// TIA Portal project "Fase_4" (V17)

(* hardware
DEVICE "S7-1200 station_1"  S7-1200 Station
   slot 0: "Rack_0"  S7-1200 Rack  Rack  V1.0
   slot 1: "PLC_1"  CPU 1214C AC/DC/Rly  6ES7 214-1BE30-0XB0  V2.2
*)

// ===== PLC "PLC_1"  CPU 1214C AC/DC/Rly =====

VAR_GLOBAL   // PLC tag table "Default tag table"
   "aumentarcoches" AT %M100.0 : Bool;
   "quitarcoches" AT %M100.1 : Bool;
   "Tag_1" AT %M202.2 : Bool;
   "Tag_2" AT %MW320 : Int;
   "Tag_3" AT %MW420 : Int;
   "verde" AT %M1.0 : Bool;
   "naranja" AT %M1.1 : Bool;
   "rojo" AT %M1.2 : Bool;
END_VAR

// folder: System blocks/Program resources

DATA_BLOCK "numerocoches"   // DB1
{ S7_Optimized_Access := 'TRUE' }
AUTHOR : Simatic
FAMILY : IEC
NAME : CNTR
VERSION : 1.0
// stored: InstanceOfName IEC_COUNTER
"IEC_COUNTER"
BEGIN
END_DATA_BLOCK

// folder: (top level)

ORGANIZATION_BLOCK "Main"   // OB1, LAD, ProgramCycle
TITLE = "Main Program Sweep (Cycle)"
{ S7_Optimized_Access := 'TRUE' }
VERSION : 0.1
// Es un garaje monitorizado.
BEGIN

REGION Network 1
   // Esto es un contador de coches, M100 aumenta en uno el numero de coches, M100.1 quita un coche y MW320  recoge el numero de coches
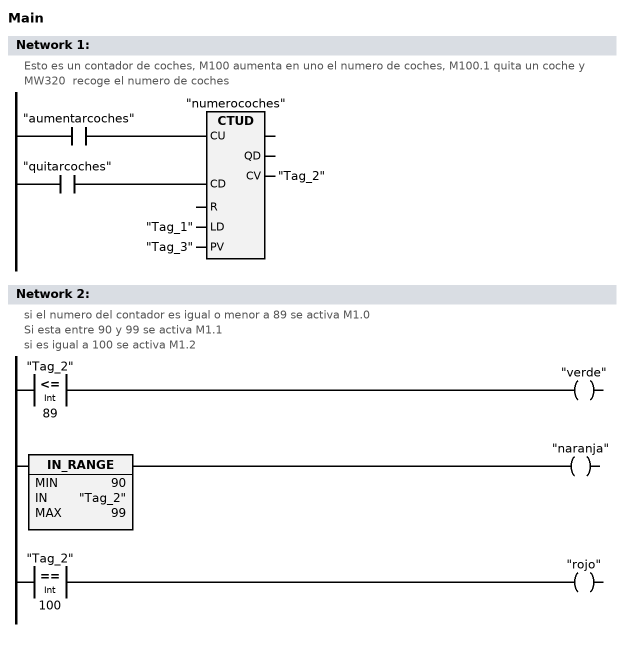
   "numerocoches".CTUD(CU := "aumentarcoches",
                       CD := "quitarcoches",
                       LD := "Tag_1",
                       PV := "Tag_3",
                       CV => "Tag_2");
END_REGION

REGION Network 2
   // si el numero del contador es igual o menor a 89 se activa M1.0
   // Si esta entre 90 y 99 se activa M1.1
   // si es igual a 100 se activa M1.2
   RUNG wire#powerrail
      { S7_Templates := "SrcType := Int" } LE_Contact(in1 := "Tag_2", in2 := 89)
      Coil( "verde" )
   END_RUNG
   RUNG wire#powerrail
      { S7_Templates := "SrcType := Int" } InRange(min := 90, in := "Tag_2", max := 99)
      Coil( "naranja" )
   END_RUNG
   RUNG wire#powerrail
      { S7_Templates := "SrcType := Int" } EQ_Contact(in1 := "Tag_2", in2 := 100)
      Coil( "rojo" )
   END_RUNG
   // the same network as SCL:
   "verde" := "Tag_2" <= 89;
   "naranja" := (90 <= "Tag_2") AND ("Tag_2" <= 99);
   "rojo" := "Tag_2" = 100;
END_REGION
END_ORGANIZATION_BLOCK